TYPE ST_Sts_PlcComIn :
STRUCT
	bSliderHomeSensor		: BOOL;
	bAngleMotorSensor		: BOOL;
	bGripperHomeSensor		: BOOL;
	PtcRawTemp				: INT;
END_STRUCT
END_TYPE

(* stored: Version 1.1.0.1
   DUT ST_Sts_PlcComIn: Id {0ec2b993-d1b9-4ec6-8253-96f008fec0fd} *)
